{attribute addProperty BoxType "EPP6001-0002-0016"}
{attribute addProperty Id "CtrlAT %Q*UINT1621Data_OutAT %Q*ARRAY[0 ..21] OF USINT176220"}
{attribute addProperty CRC "1274078981"}
{attribute addProperty SizeInBites "192"}
{attribute addProperty SizeInBytes "24"}
TYPE COM_Outputs_F536B385 :
STRUCT
	{attribute addProperty Name "Ctrl"}
	Ctrl AT %Q* : UINT;
	{attribute addProperty Name "Data_Out"}
	Data_Out AT %Q* : ARRAY[0 ..21] OF USINT;
END_STRUCT
END_TYPE

(* stored: Version 1.2.0.0, ProductVersion 3.1.4024.9
   DUT COM_Outputs_F536B385: Id {4c797bfc-91f9-4493-9310-dfbff83ac76f} *)
